FUNCTION_BLOCK PUBLIC RestorePreviousAutomaticState
VAR_INPUT
END_VAR
VAR_OUTPUT
END_VAR
VAR
	RotationRestored: BOOL := FALSE;
	LiftingRestored: BOOL := FALSE;
	ExtensionRestored: BOOL := FALSE;
	GripRestored: BOOL := FALSE;
END_VAR

// reset rotation:
IF Automatic.RotationPositionAuto - Automatic.RotationPositionCurrent > 25 THEN
	IO.MotorRotationDirection := 0;
	Automatic.MotorR.CurrentlyMoving := TRUE;
	IO.MotorRotation := 1;
ELSIF Automatic.RotationPositionCurrent - Automatic.RotationPositionAuto > 25 THEN
	IO.MotorRotationDirection := 0;
	Automatic.MotorR.CurrentlyMoving := TRUE;
	IO.MotorRotation := 1;
ELSE
	IO.MotorRotation := 0;
	Automatic.MotorR.CurrentlyMoving := FALSE;
END_IF
// reset lifting:
IF Automatic.LiftingPositionAuto - Automatic.LiftingPositionCurrent > 25 THEN
	IO.MotorLiftingDirection := 0;
	Automatic.MotorL.CurrentlyMoving := TRUE;
	IO.MotorLifting := 1;
ELSIF Automatic.LiftingPositionCurrent - Automatic.LiftingPositionAuto > 25 THEN
	IO.MotorLiftingDirection := 0;
	Automatic.MotorL.CurrentlyMoving := TRUE;
	IO.MotorLifting := 1;
ELSE
	IO.MotorLifting := 0;
	Automatic.MotorL.CurrentlyMoving := FALSE;
END_IF
// reset extension:
IF Automatic.ExtensionPositionAuto - Automatic.ExtensionPositionCurrent > 25 THEN
	IO.MotorExtensionDirection := 0;
	Automatic.MotorE.CurrentlyMoving := TRUE;
	IO.MotorExtension := 1;
ELSIF Automatic.ExtensionPositionCurrent - Automatic.ExtensionPositionAuto > 25 THEN
	IO.MotorExtensionDirection := 0;
	Automatic.MotorE.CurrentlyMoving := TRUE;
	IO.MotorExtension := 1;
ELSE
	IO.MotorExtension := 0;
	Automatic.MotorE.CurrentlyMoving := FALSE;
END_IF
// reset grip:
IF Automatic.GripPositionAuto - Automatic.GripPositionCurrent > 25 THEN
	IO.MotorGripDirection := 0;
	Automatic.MotorG.CurrentlyMoving := TRUE;
	IO.MotorGrip := 1;
ELSIF Automatic.GripPositionCurrent - Automatic.GripPositionAuto > 25 THEN
	IO.MotorGripDirection := 0;
	Automatic.MotorG.CurrentlyMoving := TRUE;
	IO.MotorGrip := 1;
ELSE
	IO.MotorGrip := 0;
	Automatic.MotorG.CurrentlyMoving := FALSE;
END_IF

// if all restored then go on to exeecute recipes in AutomaticControl:
IF RotationRestored AND LiftingRestored AND ExtensionRestored AND GripRestored THEN
	IO.SwitchedToAutomatic := FALSE;
END_IF

END_FUNCTION_BLOCK

(* stored: Version 1.1.0.1, ProductVersion 3.1.4024.13
   POU RestorePreviousAutomaticState: Id {bf2e792f-bc3c-4ce2-afd6-05125fa35279}, SpecialFunc None *)
